(* PLC project SafeLOGIC, BrAutomation SafeDESIGNER  5.24.1.0 *)
(* stored: companyURL http://www.br-automation.com, creationDateTime Sun Oct 26 13:19:39 2025 *)

PROGRAM RO_SMxxx

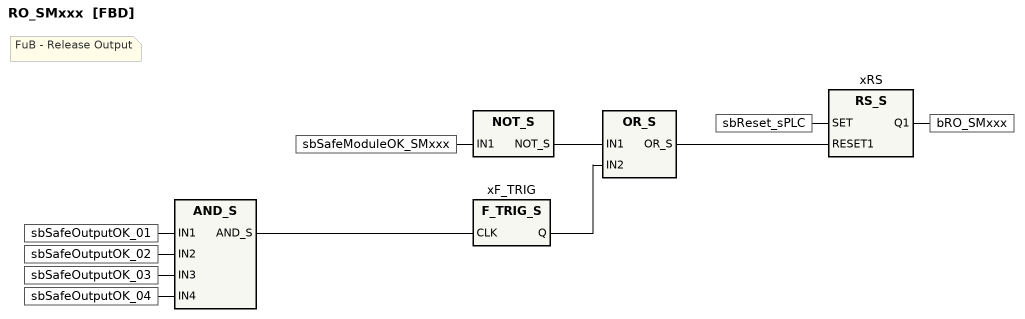
(* FBD diagram, written out as Structured Text *)
(* FuB - Release Output *)
xF_TRIG(CLK := AND_S(sbSafeOutputOK_01, sbSafeOutputOK_02, sbSafeOutputOK_03, sbSafeOutputOK_04));
xRS(SET := sbReset_sPLC, RESET1 := OR_S(NOT_S(sbSafeModuleOK_SMxxx), xF_TRIG.Q));
bRO_SMxxx := xRS.Q1;
END_PROGRAM
